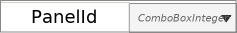
VISUALIZATION V_PanelSelecCmb  // 237x33
    ComboBoxInteger (129,3 108x30), variable: VisuGVL.fbPanelImp.PanelId, text list: 'PanelCmbTxtList'
    Textfield (0,2 129x30), "PanelId"
END_VISUALIZATION

(* stored: Version 1.1.0.1, ProductVersion 3.1.4024.4
   Visu V_PanelSelecCmb: Id {806a373f-b841-449f-9dbd-3c0278f46dd7} *)
